Omron CX-Programmer project NewProject (CX-Programmer 9.61)

# PLC PLC_Water_Treatment_Control: CJ2M CPU11

## Global symbols (name address type ; comment)
0.00 BOOL  ; P_Start
0.01 BOOL  ; Emergency
0.02 BOOL  ; Manual_mode
0.03 BOOL  ; Reset
0.04 BOOL  ; P_Water_Pump
0.05 BOOL  ; P_Alkaline_Pump
0.06 BOOL  ; P_Acid_Pump
0.07 BOOL  ; P_reset
0.08 BOOL  ; Max_Water_Sensor
0.09 BOOL  ; Output_Valve
0.10 BOOL  ; P_Stop
0.11 BOOL  ; a
100.00 BOOL  ; Start
100.01 BOOL  ; Water_Pump
100.02 BOOL  ; Alkaline_Pump
100.03 BOOL  ; Acid_Pump
100.04 BOOL  ; Max_Level
100.05 BOOL  ; Mid_level
100.06 BOOL  ; Empty
100.07 BOOL  ; Valve
100.08 BOOL  ; Manual
D100 CHANNEL  ; Water
D101 CHANNEL  ; pH
D200 CHANNEL  ; HMI_Water_Level
D201 CHANNEL  ; HDMI_pH_Level

## Program NewProgram1 (cyclic task 0)

### Section Section1

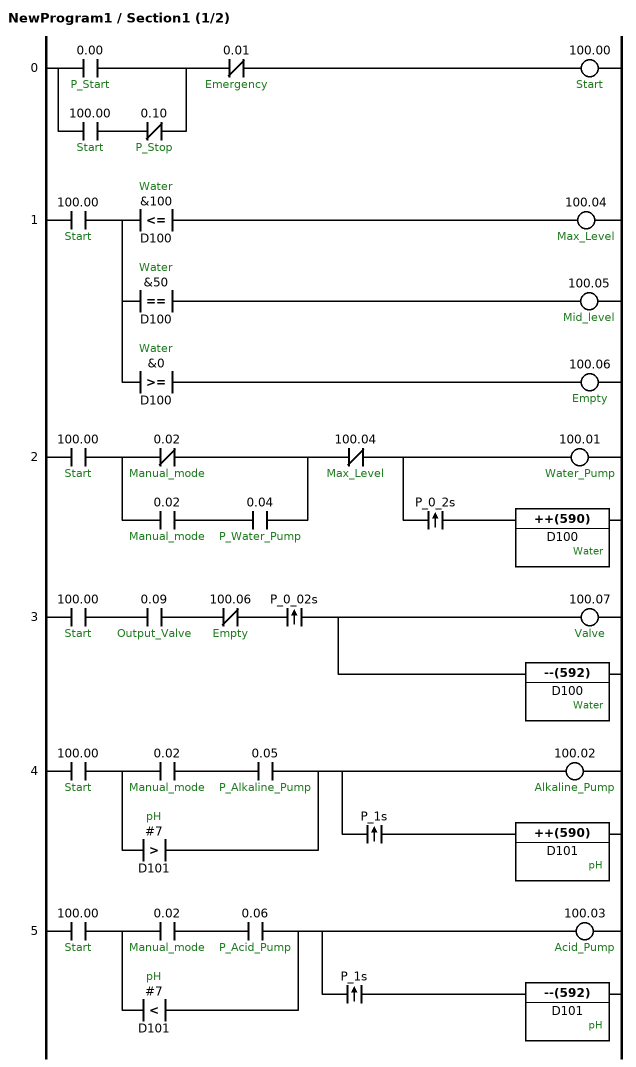
; rung 0
LD 0.00  ; P_Start
LD 100.00  ; Start
ANDNOT 0.10  ; P_Stop
ORLD
ANDNOT 0.01  ; Emergency
OUT 100.00  ; Start
; rung 1
LD 100.00  ; Start
OUT TR0
AND<=(315) &100 D100  ; Water
OUT 100.04  ; Max_Level
LD TR0
AND=(300) &50 D100  ; Water
OUT 100.05  ; Mid_level
LD TR0
AND>=(325) &0 D100  ; Water
OUT 100.06  ; Empty
; rung 2
LD 100.00  ; Start
LDNOT 0.02  ; Manual_mode
LD 0.02  ; Manual_mode
AND 0.04  ; P_Water_Pump
ORLD
ANDLD
ANDNOT 100.04  ; Max_Level
OUT 100.01  ; Water_Pump
@AND P_0_2s
++(590) D100  ; Water
; rung 3
LD 100.00  ; Start
AND 0.09  ; Output_Valve
ANDNOT 100.06  ; Empty
@AND P_0_02s
OUT 100.07  ; Valve
--(592) D100  ; Water
; rung 4
LD 100.00  ; Start
LD 0.02  ; Manual_mode
AND 0.05  ; P_Alkaline_Pump
OR>(320) #7 D101  ; pH
ANDLD
OUT 100.02  ; Alkaline_Pump
@AND P_1s
++(590) D101  ; pH
; rung 5
LD 100.00  ; Start
LD 0.02  ; Manual_mode
AND 0.06  ; P_Acid_Pump
OR<(310) #7 D101  ; pH
ANDLD
OUT 100.03  ; Acid_Pump
@AND P_1s
--(592) D101  ; pH

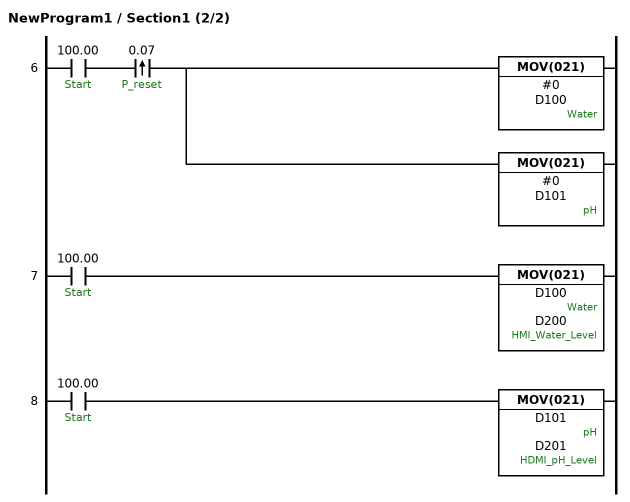
; rung 6
LD 100.00  ; Start
@AND 0.07  ; P_reset
MOV(021) #0 D100  ; Water
MOV(021) #0 D101  ; pH
; rung 7
LD 100.00  ; Start
MOV(021) D100 D200  ; Water, HMI_Water_Level
; rung 8
LD 100.00  ; Start
MOV(021) D101 D201  ; pH, HDMI_pH_Level

### Section END
; rung 0
END(001)